// TIA Portal V17 export
// export: Created 2025-03-05T08:01:43.2466558Z, ExportSetting WithDefaults, DisplayName Totally Integrated Automation Portal, DisplayVersion V17 Update 8, DisplayName TIA Portal Openness, DisplayVersion V17 Update 8, DisplayName TIA Portal Version Control Interface, DisplayVersion V17, DisplayName SINAMICS Startdrive Advanced, DisplayVersion V17 SP2, DisplayName SINAMICS Startdrive G110M, G120, G120C, G120D, G120P, G115D, DisplayVersion V17 SP2, DisplayName SINAMICS Startdrive G130, G150, S120, S150, SINAMICS MV, S210, DisplayVersion V17 SP2, DisplayName STEP 7 Professional, DisplayVersion V17 Update 8, DisplayName SINUMERIK ONE STEP 7 Toolbox, DisplayVersion V17 Update 12, DisplayName SINUMERIK 840D sl STEP 7 Toolbox, DisplayVersion V17 Update 12, DisplayName STEP 7 Safety, DisplayVersion V17 Update 6, DisplayName WinCC Advanced, DisplayVersion V17 Update 8
DATA_BLOCK "DB7227_24_HOURS_TEST"   // DB7227
{ S7_Optimized_Access := 'FALSE'; DB_Accessible_From_OPC_UA := 'FALSE' }
AUTHOR : ETXETAR
VERSION : 1.0
// stored: AutoNumber false, DBAccessibleFromOPCUA false, DBAccessibleFromWebserver true, IsOnlyStoredInLoadMemory false, IsWriteProtectedInAS false
   VAR RETAIN
      TEST24H_START_REQ : Bool;   // TEST24H START REQ
      TEST24H_SCRIPT : Bool;   // TEST24H SCRIPT
      TEST24H_TEST_DONE : Bool;   // TEST24H TEST DONE
      TEST24H_START_REQ_AUX : Bool;   // TEST24H START REQ AUX
      TEST24H_TEST_DONE_AUX : Bool;   // TEST24H TEST DONE AUX
      TEST24H_XFLEX_XFLEX_DUO : Bool;   // TEST24H XFLEX XFLEX DUO
      TEST24H_SEOC_AFTER_DONE : Bool;   // TEST24H SEOC AFTER DONE
      TEST24H_RESET_TEST_DONE : Bool;   // TEST24H RESET TEST DONE
      TEST24H_TCU_PCU : Bool;   // TEST24H TCU PCU
      TEMP_DATA { S7_SetPoint := 'True'} : "TEST_24HRS";   // TEMP DATA
      TIMER_24H_AUX { S7_SetPoint := 'True'} : TON_TIME;   // TIMER 24H AUX
   END_VAR
BEGIN
   TIMER_24H_AUX.PT := T#48H;
END_DATA_BLOCK
